// TIA Portal V17 export
// export: Created 2022-04-06T07:28:39.9230363Z, ExportSetting WithDefaults, DisplayName Totally Integrated Automation Portal, DisplayVersion V17, DisplayName TIA Portal Openness, DisplayVersion V17, DisplayName TIA Portal Version Control Interface, DisplayVersion V17, DisplayName TIA Portal Test Suite Advanced, DisplayVersion V17, DisplayName SINAMICS Startdrive Advanced, DisplayVersion V17, DisplayName SINAMICS Startdrive G130, G150, S120, S150, SINAMICS MV, S210, DisplayVersion V17, DisplayName SINAMICS Startdrive G110M, G120, G120C, G120D, G120P, G115D, DisplayVersion V17, DisplayName STEP 7 Professional, DisplayVersion V17, DisplayName STEP 7 Safety, DisplayVersion V17, DisplayName WinCC Advanced / Unified PC, DisplayVersion V17
DATA_BLOCK "InstTestSCL"   // DB8
VERSION : 0.1
// stored: AutoNumber true, DBAccessibleFromOPCUA true, DBAccessibleFromWebserver true, InstanceOfName TestSCL, InstanceOfType FB
"TestSCL"
   // VAR_INPUT
   //    start : Bool;
   //    stop : Bool;
   // END_VAR
   // VAR_OUTPUT
   //    valueIsReached : Bool;
   //    currentValue : Int;
   //    run : Bool;
   // END_VAR
   // VAR
   //    instRTrigForRun { S7_SetPoint := 'True'} : R_TRIG;
   //    startRisingEdge : Bool;
   // END_VAR
   // VAR RETAIN
   //    instCounterAdd1 { S7_SetPoint := 'True'} : CTU_INT;
   //    IEC_Counter_0_Instance { S7_SetPoint := 'True'} : CTU_INT;
   //    statState { S7_SetPoint := 'True'} : DInt;
   // END_VAR
   // VAR
   //    instRTrig { S7_SetPoint := 'True'} : R_TRIG;
   //    instLGF_FIFO { S7_SetPoint := 'True'} : "LGF_FIFO";
   //    statCount { S7_SetPoint := 'True'} : Int;
   //    statLogFileName : String[50];
   //    statlogFileNameTemp : Array[0..10] of String[50];
   // END_VAR
BEGIN
END_DATA_BLOCK
